INTERFACE I_HostSynchronousRpcHandlers

METHOD PUBLIC RegisterHandler
VAR_INPUT
	MethodName : T_MAXSTRING;
	Handler : I_SynchronousRpcHandler;
END_VAR
END_METHOD

END_INTERFACE

(* stored: Version 1.1.0.1, ProductVersion 3.1.4026.13
   Itf I_HostSynchronousRpcHandlers: Id {4dc47ead-7e95-013b-17c1-849edaed8fde}
   Method RegisterHandler: Id {b394f5c7-3815-0bfb-1de1-d19473e24487} *)
